
// ===== library types =====

TYPE "UDT_AO"
   STRUCT
      In : Real;   // Входное значение для вывода
      Par_max : Real := 100.0;   // Максимальное значение шкалы
      Par_min : Real;   // Минимальное занчение шкалы
      RezCh : Bool;   // В true если канал резервный
      Out : Int;   // Обработанное занчение на выход модуля
   END_STRUCT;
END_TYPE

TYPE "UDT_DI"
VERSION : 0.1
   STRUCT
      ReservChannel : Bool;   // Признак резервного бита
      Value : Bool;   // Выходное значение
      Invert : Bool;   // Инверсия
      In_Value : Bool;   // Входное значение
      Simulate : Bool;   // Симуляция
      Sim_Value : Bool;   // Значение симуляции
   END_STRUCT;
END_TYPE

TYPE "UDT_AI"
VERSION : 0.1
   STRUCT
      Raw_in : Int;   // Код АЦП - входное значение с модуля / Входной сигнал от модуля
      Out_value : Real;   // Масштабированное значение / Выходной преобразованный сигнал
      Field_value : Real;   // Значение тока (напряжения) с датчика
      Value_hi_scale : Int := 100;   // Максимальное физическое значение / Верняя шкала
      Value_lo_scale : Int;   // Минимальное физическое значение / Нижняя жкала
      Hihi_limit : Real;   // Значение верхней аварийной границы / ВАУ
      Hi_limit : Real;   // Значение верхней предупредительной границы / ВПУ
      Lo_limit : Real;   // Значение нижней предупредительной границы / НПУ
      Lolo_limit : Real;   // Значение нижней аварийной границы / НАУ
      Simulate_In : Real;   // Заданное значение симуляции / Значение симуляции
      Raw_lo_scale : Int := 5530;   // Код АЦП - нижняя граница значения
      Raw_hi_scale : Int := 27648;   // Код АЦП - верхняя граница значения
      Raw_lo_error : Int := 4838;   // Код АЦП - граница обрыва
      Raw_hi_error : Int := 28000;   // Код АЦП - граница короткого замыкания
      Field_lo_scale : Real := 4.0;   // Минимальное значение тока (напряжения)
      Field_hi_scale : Real := 20.0;   // Максимальное значение тока (напряжения)
      Digital_in : Real;   // Входное масштабированное значение
      RezervChannel : Bool;   // Признак резервного канала
      En_Digital_in : Bool;   // Разрешение - вход для значения Real вместо Int (Word)
      Simulate : Bool;   // Разрешение - режим симуляции / Признак цимуляции
      Hihi_enable : Bool;   // Разрешение - обработка сигнала Hihi / Активация ВАУ
      Hi_enable : Bool;   // Разрешение - обработка сигнала Hi / Активация ВПУ
      Lo_enable : Bool;   // Разрешение - обработка сигнала Lo / Активация НПУ
      Lolo_enable : Bool;   // Разрешение - обработка сигнала Lolo / Активация НАУ
      Hihi_act : Bool;   // Флаг - значение в верхней аварийной зоне / Сработка ВАУ
      Hi_act : Bool;   // Флаг - значение в верхней предупредительной зоне / Сработка ВПУ
      Lo_act : Bool;   // Флаг - значение в верхней предупредительной зоне / Сработка НПУ
      Lolo_act : Bool;   // Флаг - значение в нижней аварийной зоне / Сработка НАУ
      Lo_raw : Bool;   // Флаг - обрыв / Обрыв
      Hi_raw : Bool;   // Флаг - короткое замыкание / КЗ
      Alarm : Bool;   // Флаг - значение в аварийной зоне / Авария
      Warning : Bool;   // Флаг - значение в предупредительной зоне / Предупреждение
      Nominal : String := 'mm';   // Размерность един. изм.
   END_STRUCT;
END_TYPE

TYPE "UDT_IM"
   STRUCT
      SO : Bool;   // Состояние вкл/открыто
      SC : Bool;   // Состояние откл/закрыто
      SA : Bool;   // Состояние авария
      DU : Bool;   // Состояние дистанционное управление
      MU : Bool;   // Состояние местное управление
      Q_CO : Bool;   // Команда вкл/открыть
      Q_CS : Bool;   // Команда откл/закрыть
      B_CO : Bool;   // Команда открыть/вклюсить по алгоритму
      B_CS : Bool;   // Команда закрыть/выключить по алгоритму
      HMI_CO : Bool;   // Команда открыть/включить от ВУ
      HMI_CS : Bool;   // Команда закрыть/отключить от ВУ
      I_REP : Bool;   // Команда ремонт
      Q_REP : Bool;   // Выход команды ремонт
      Load : Int;   // Значение нагрузки
      TON_PT : Time := T#60000ms;
      TON_ET : Time;
      TON_IN : Bool;
      TON_Q : Bool;
   END_STRUCT;
END_TYPE

// folder: AI

FUNCTION "Proc_AI" : Void   // FC100, SCL
{ S7_Optimized_Access := 'TRUE' }
AUTHOR : SybCom
VERSION : 0.1
   VAR_TEMP
      i : Int;
      j : Int;
      Out_scaled : Real;
      AVG_Value : Real;
      Summ_Massive : Real;
      Result : Int;
      NumAnalog : Int;
      Dtl_now : DTL;
      One_sec_on : Bool;
      H_msec_on : Bool;
      AI_ACP_REAL : Real;
      MAX_ACP_REAL : Real;
      MIN_ACP_REAL : Real;
   END_VAR
BEGIN
   //AUTHOR: frozi2
   //DESC: Блок входного аналогового сигнала

   // Блок инициализации данных
   //2A1.3
   (*
   "Data_AI".Data[1].Raw_in := "AI1";//"PT-10"; //Давление сжатого воздуха
   "Data_AI".Data[2].Raw_in := "AI2";//"PT-01"; //Разрежение до РФ
   "Data_AI".Data[3].Raw_in := "AI3";//"PT-02"; //Разрежение после РФ
   "Data_AI".Data[4].Raw_in := "TT-01"; //Температура газа перед клапаном ав. подсоса
   "Data_AI".Data[5].Raw_in := "TT-02"; //Температура газа перед РФ
   "Data_AI".Data[6].Raw_in := "QT-101"; //Запыленность газа
   "Data_AI".Data[7].Raw_in := "FT-101"; //Расход газа
   "Data_AI".Data[8].Raw_in := "TT-03"; //Температура газа на выходе
   *)
   //2A1.4
   //"Data_AI".Data[9].Raw_in  := "2A1_4_AI_00"; //Давление воды 
   //"Data_AI".Data[10].Raw_in := "2A1_4_AI_01"; //Давление до 
   //"Data_AI".Data[11].Raw_in := "2A1_4_AI_02"; //Давление после 
   //"Data_AI".Data[12].Raw_in := "2A1_4_AI_03"; //Резерв
   //"Data_AI".Data[13].Raw_in := "2A1_4_AI_04"; //Резерв
   //"Data_AI".Data[14].Raw_in := "2A1_4_AI_05"; //Резерв
   //"Data_AI".Data[15].Raw_in := "2A1_4_AI_06"; //Резерв
   //"Data_AI".Data[16].Raw_in := "2A1_4_AI_07"; //Резерв
   (*
   FOR #i := 1 TO "Data_AI".Num_AI DO
       IF (#i > 4 AND #i < 9) OR #i > 11 THEN
           "Data_AI".Data[#i].RezervChannel := TRUE;
       ELSE
           "Data_AI".Data[#i].RezervChannel := FALSE;
       END_IF;
   END_FOR;
   *)

   //для расшифровки кода АЦП


   // Обработка сигналов
   FOR #i := 1 TO "Data_AI".Num_AI DO
     // Если канал не резервный
       IF NOT "Data_AI".Data[#i].RezervChannel THEN

           // Приведение к другому типу для удобства вычислений
           #AI_ACP_REAL := DINT_TO_REAL(WORD_TO_DINT("Data_AI".Data[#i].Raw_in));   // Перевод из WORD в REAL значение с АЦП входа
           #MAX_ACP_REAL := DINT_TO_REAL(WORD_TO_DINT("Data_AI".Data[#i].Value_hi_scale)); // Перевод из WORD в REAL Шкалы макс.
           #MIN_ACP_REAL := DINT_TO_REAL(WORD_TO_DINT("Data_AI".Data[#i].Value_lo_scale)); // Перевод из WORD в REAL Шкалы мин.

           //Масштабирование величин
           //Токовое значение с датчика   
           "Data_AI".Data[#i].Field_value := (("Data_AI".Data[#i].Field_hi_scale - "Data_AI".Data[#i].Field_lo_scale) / ("Data_AI".Data[#i].Raw_hi_scale - "Data_AI".Data[#i].Raw_lo_scale)) *
           ("Data_AI".Data[#i].Raw_in - "Data_AI".Data[#i].Raw_lo_scale) + "Data_AI".Data[#i].Field_lo_scale;

           //Физическое значение с датчика
           #Out_scaled := (#MAX_ACP_REAL - #MIN_ACP_REAL) / ("Data_AI".Data[#i].Raw_hi_scale - "Data_AI".Data[#i].Raw_lo_scale) *
           (#AI_ACP_REAL - "Data_AI".Data[#i].Raw_lo_scale) + #MIN_ACP_REAL;



       // Полученный сигнал уже масштабирован
       IF "Data_AI".Data[#i].En_Digital_in THEN
         #Out_scaled := "Data_AI".Data[#i].Digital_in;
       END_IF;
       // Симуляция выходной величины
       IF "Data_AI".Data[#i].Simulate THEN
         #Out_scaled := "Data_AI".Data[#i].Simulate_In;
       END_IF;
       // Усреднение и нижняя отсечка (удалено из DB)    
       (*  

       //Запоминание времени
       #Result := RD_LOC_T(#Dtl_now);
       //Счетчик для усреднения величины
       if TOD_TO_DINT(DTL_TO_TOD(#Dtl_now)) - TOD_TO_DINT(DTL_TO_TOD("DataHelpAI".Data[i].Dtl_h_msec)) >
          INT_TO_DINT("DataHelpAI".Data[i].Bal_time) * 100 then
         #H_msec_on := True;
       end_if;
       //Усреднение величины ведется с кратностью в 100 мс.
       if #H_msec_on then
         #Result := RD_LOC_T("DataHelpAI".Data[i].Dtl_h_msec);
         #H_msec_on := False;
         //Запись в массив ведется циклично
         "DataHelpAI".Data[i].Massive_point := "DataHelpAI".Data[i].Massive_point + 1;  
         if "DataHelpAI".Data[i].Massive_point > 9 then
           "DataHelpAI".Data[i].Massive_point := 0;
         end_if;
         //Сохранение величины в массиве
         "DataHelpAI".Data[i].Output_Massive["DataHelpAI".Data[i].Massive_point] := #Out_scaled;  
       end_if;
       #AVG_Value := 0;
       if "DataHelpAI".Data[i].Bal_time > 0 then
         #Summ_Massive := 0;
         for #j := 0 to 9 do
           #Summ_Massive := #Summ_Massive + "DataHelpAI".Data[i].Output_Massive[#j];
         end_for;
         #AVG_Value := #Summ_Massive / 10;
         #Out_scaled := #AVG_Value;
       end_if;
       //Проверка на зону нечувствительности 
       if ABS("DataHelpAI".Data[i].Previos_val - #Out_scaled) < "DataHelpAI".Data[i].Value_db then
         #Out_scaled := "DataHelpAI".Data[i].Previos_val;
       end_if;
       //Проверка на нижнюю отсечку  
       if (#Out_scaled < "DataHelpAI".Data[i].Lo_cutoff) & "DataHelpAI".Data[i].Lo_cut_enable then
         #Out_scaled := "DataHelpAI".Data[i].Lo_cutoff;
       end_if;
   *)



       // Формирование аварий  
       // Обрыв  
       IF ("Data_AI".Data[#i].Raw_in <= "Data_AI".Data[#i].Raw_lo_error) AND
         NOT "Data_AI".Data[#i].Simulate THEN
         "Data_AI".Data[#i].Lo_raw := True;
         #Out_scaled := "Data_AI".Data[#i].Value_lo_scale;
       ELSE
         "Data_AI".Data[#i].Lo_raw := False;
       END_IF;

       // КЗ датчика
       IF ("Data_AI".Data[#i].Raw_in >= "Data_AI".Data[#i].Raw_hi_error) AND
         NOT "Data_AI".Data[#i].Simulate THEN
         "Data_AI".Data[#i].Hi_raw := True;
         #Out_scaled := "Data_AI".Data[#i].Value_hi_scale;
       ELSE
         "Data_AI".Data[#i].Hi_raw := False;
       END_IF;

       // Нижняя аварийная зона
       IF #Out_scaled < "Data_AI".Data[#i].Lolo_limit AND
           "Data_AI".Data[#i].Lolo_enable AND NOT "Data_AI".Data[#i].Lo_raw THEN
           "Data_AI".Data[#i].Lolo_act := True;
       ELSE
           "Data_AI".Data[#i].Lolo_act := False;
       END_IF;

       // Нижняя предупредительная зона
       IF #Out_scaled < "Data_AI".Data[#i].Lo_limit AND NOT "Data_AI".Data[#i].Lolo_act AND
           "Data_AI".Data[#i].Lo_enable AND NOT "Data_AI".Data[#i].Lo_raw THEN
           "Data_AI".Data[#i].Lo_act := True;
       ELSE
           "Data_AI".Data[#i].Lo_act := False;
       END_IF;
       // Верхняя предупредительная зона
       IF #Out_scaled > "Data_AI".Data[#i].Hi_limit AND NOT "Data_AI".Data[#i].Hihi_act AND
           "Data_AI".Data[#i].Hi_enable AND NOT "Data_AI".Data[#i].Hi_raw THEN
           "Data_AI".Data[#i].Hi_act := True;
       ELSE
           "Data_AI".Data[#i].Hi_act := False;
       END_IF;

       // Верхняя аварийная зона
       IF #Out_scaled > "Data_AI".Data[#i].Hihi_limit AND
           "Data_AI".Data[#i].Hihi_enable AND NOT "Data_AI".Data[#i].Hi_raw THEN
           "Data_AI".Data[#i].Hihi_act := True;
       ELSE
           "Data_AI".Data[#i].Hihi_act := False;
       END_IF;

       // Определение флага предупреждения
       IF ("Data_AI".Data[#i].Hi_act OR "Data_AI".Data[#i].Lo_act) THEN
         "Data_AI".Data[#i].Warning := true;
       ELSE
         "Data_AI".Data[#i].Warning := false;
       END_IF;

       // Определение флага аварии
       IF "Data_AI".Data[#i].Hihi_act OR "Data_AI".Data[#i].Lolo_act  THEN
         "Data_AI".Data[#i].Alarm := true;
       ELSE
         "Data_AI".Data[#i].Alarm := false;
       END_IF;

       // Сохранение значения
       "Data_AI".Data[#i].Out_value := #Out_scaled;
     END_IF;
   END_FOR;
END_FUNCTION

// folder: AO

FUNCTION "Proc_AO" : Void   // FC102, SCL
{ S7_Optimized_Access := 'TRUE' }
VERSION : 0.1
   VAR_TEMP
      i : Int;
      Temp_out : Real;
   END_VAR
BEGIN
   //AUTHOR: frozi2
   //DESC: Блок выходного аналогового сигнала

   // Блок инициализации данных
   //2A1.3
   "Data_AO".Data[1].In := "AI1";//"PT-10"; //Давление сжатого воздуха
   "Data_AO".Data[2].In := "AI2";//"PT-01"; //Разрежение до РФ
   "Data_AO".Data[3].In := "AI3";//"PT-02"; //Разрежение после РФ
   "Data_AO".Data[4].In := "TT-01"; //Температура газа перед клапаном ав. подсоса
   "Data_AO".Data[5].In := "TT-02"; //Температура газа перед РФ
   "Data_AO".Data[6].In := "QT-101"; //Запыленность газа
   "Data_AO".Data[7].In := "FT-101"; //Расход газа
   "Data_AO".Data[8].In := "TT-03"; //Температура газа на выходе


   //Задействовать это часть для анализа резервных каналов и исключения их их опроса или принудительно
   //устанавливать переменную RezervChannel = 1, в Data_AO для каждого резервного канала
   (*
   FOR #i := 1 TO "Data_AI".Num_AO DO
       IF (#i > 4 AND #i < 9) OR #i > 11 THEN  //тут отредактировать по своим условиям
           "Data_AO".Data[#i].RezCh := TRUE;
       ELSE
           "Data_A0".Data[#i].RezCh := FALSE;
       END_IF;
   END_FOR;
   *)

   // Обработка сигналов
   FOR #i := 1 TO "Data_AO".Num_AO DO

       #Temp_out := ((27648.0 - 0.0)*("Data_AO".Data[#i].In - "Data_AO".Data[#i].Par_min))/("Data_AO".Data[#i].Par_max - "Data_AO".Data[#i].Par_min);

       // Если канал не резервный
       IF NOT "Data_AO".Data[#i].RezCh THEN

           // Сохранение значения
           "Data_AO".Data[#i].Out := DINT_TO_INT(REAL_TO_DINT(#Temp_out));

       END_IF;

   END_FOR;
END_FUNCTION

// folder: DI

FUNCTION "Proc_DI" : Void   // FC101, SCL
{ S7_Optimized_Access := 'TRUE' }
AUTHOR : SybCom
VERSION : 0.1
   VAR_TEMP
      i : Int;
      j : Int;
      TempValue : Bool;
      H_msec_on : Bool;
      Result : Int;
      Dtl_now : DTL;
      Summ_Massive : Real;
   END_VAR
BEGIN
   //AUTHOR: frozi2
   //DESC: Блок дискретного сигнала

   // Блок инициализации данных
   // 2A1
   "Data_DI".Data[1].In_Value := "LSA-11";  //Минимальный уровень бункера 1
   "Data_DI".Data[2].In_Value := "LSA-12";  //Верхний уровень бункера 1
   "Data_DI".Data[3].In_Value := "LSA-13";  //Минимальный уровень бункера 2
   "Data_DI".Data[4].In_Value := "LSA-14";  //Верхний уровень бункера 2
   "Data_DI".Data[5].In_Value := "LSA-15";  //Минимальный уровень бункера 3
   "Data_DI".Data[6].In_Value := "LSA-16";  //Верхний уровень бункера 3
   "Data_DI".Data[7].In_Value := "LSA-17";  //Минимальный уровень бункера 4
   "Data_DI".Data[8].In_Value := "LSA-18";  //Верхний уровень бункера 4
   "Data_DI".Data[9].In_Value := 0;  //Резерв
   "Data_DI".Data[10].In_Value := 0; //Резерв
   "Data_DI".Data[11].In_Value := 0; //Резерв
   "Data_DI".Data[12].In_Value := 0; //Резерв
   "Data_DI".Data[13].In_Value := 0; //Резерв
   "Data_DI".Data[14].In_Value := 0; //Резерв
   (*
   //2A1.5
   "Data_DI".Data[15].In_Value := "2A1_5_DI_00"; //Зд1 поз.7.2 - Открыта
   "Data_DI".Data[16].In_Value := "2A1_5_DI_01"; //Зд1 поз.7.2 - Закрыта
   "Data_DI".Data[17].In_Value := "2A1_5_DI_02"; //Зд1 поз.7.2 - Неисправность
   "Data_DI".Data[18].In_Value := "2A1_5_DI_03"; //Зд2 поз.7.2 - Открыта
   "Data_DI".Data[19].In_Value := "2A1_5_DI_04"; //Зд2 поз.7.2 - Закрыта
   "Data_DI".Data[20].In_Value := "2A1_5_DI_05"; //Зд2 поз.7.2 - Неисправность
   "Data_DI".Data[21].In_Value := "2A1_5_DI_06"; //Зд3 поз.7.2 - Открыта
   "Data_DI".Data[22].In_Value := "2A1_5_DI_07"; //Зд3 поз.7.2 - Закрыта
   "Data_DI".Data[23].In_Value := "2A1_5_DI_08"; //Зд3 поз.7.2 - Неисправность
   "Data_DI".Data[24].In_Value := "2A1_5_DI_09"; //УПОУ поз.7.2 - Исправен 1к
   "Data_DI".Data[25].In_Value := "2A1_5_DI_10"; //УПОУ поз.7.2 - ВТО 1к
   "Data_DI".Data[26].In_Value := "2A1_5_DI_11"; //Резерв
   "Data_DI".Data[27].In_Value := "2A1_5_DI_12"; //С2000-СП1 №1 - «Пожар в блоке» - поз.2.3
   "Data_DI".Data[28].In_Value := "2A1_5_DI_13"; //С2000-СП1 №1 - «Пожар в блоке» - поз.3.2
   "Data_DI".Data[29].In_Value := "2A1_5_DI_14"; //С2000-СП1 №1 - «Пожар в блоке» - поз.6.3(1)
   "Data_DI".Data[30].In_Value := "2A1_5_DI_15"; //С2000-СП1 №1 - «Пожар в блоке» - поз.6.3(2)

   //2A1.6
   "Data_DI".Data[31].In_Value := "2A1_6_DI_00"; //С2000-СП1 №2 - «Пожар»
   "Data_DI".Data[32].In_Value := "2A1_6_DI_01"; //С2000-СП1 №2 - «Неисправность»
   "Data_DI".Data[33].In_Value := "2A1_6_DI_02"; //Резерв
   "Data_DI".Data[34].In_Value := "2A1_6_DI_03"; //Резерв
   "Data_DI".Data[35].In_Value := "2A1_6_DI_04"; //Сигнал 20П - Несанкционированный вход
   "Data_DI".Data[36].In_Value := "2A1_6_DI_05"; //Сигнал 20П - Неисправность
   "Data_DI".Data[37].In_Value := "2A1_6_DI_06"; //Шкаф ШОС - Обобщенный сигнал несанкционированного входа
   "Data_DI".Data[38].In_Value := "2A1_6_DI_07"; //Шкаф ШОС - Неисправность
   "Data_DI".Data[39].In_Value := "2A1_6_DI_08"; //Состояние ЭЦН скважины 1.25
   "Data_DI".Data[40].In_Value := "2A1_6_DI_09"; //Состояние ЭЦН скважины 1.26
   "Data_DI".Data[41].In_Value := "2A1_6_DI_10"; //Состояние ЭЦН скважины 1.27
   "Data_DI".Data[42].In_Value := "2A1_6_DI_11"; //Состояние ЭЦН скважины 1.28
   "Data_DI".Data[43].In_Value := "2A1_6_DI_12"; //Состояние ЭЦН скважины 1.29
   "Data_DI".Data[44].In_Value := "2A1_6_DI_13"; //Состояние ЭЦН скважины 1.30
   "Data_DI".Data[45].In_Value := "2A1_6_DI_14"; //Состояние ЭЦН скважины 1.31
   "Data_DI".Data[46].In_Value := "2A1_6_DI_15"; //Состояние ЭЦН скважины 1.32

   //2A1.7
   "Data_DI".Data[47].In_Value := "2A1_7_DI_00"; //Состояние ЭЦН скважины 1.33
   "Data_DI".Data[48].In_Value := "2A1_7_DI_01"; //Состояние ЭЦН скважины 1.34
   "Data_DI".Data[49].In_Value := "2A1_7_DI_02"; //Состояние ЭЦН скважины 1.35
   "Data_DI".Data[50].In_Value := "2A1_7_DI_03"; //Состояние ЭЦН скважины 1.36
   "Data_DI".Data[51].In_Value := "2A1_7_DI_04"; //Состояние ЭЦН скважины 1.37
   "Data_DI".Data[52].In_Value := "2A1_7_DI_05"; //Состояние ЭЦН скважины 1.38
   "Data_DI".Data[53].In_Value := "2A1_7_DI_06"; //Состояние ЭЦН скважины 1.39
   "Data_DI".Data[54].In_Value := "2A1_7_DI_07"; //Состояние ЭЦН скважины 1.40
   "Data_DI".Data[55].In_Value := "2A1_7_DI_08"; //Состояние ЭЦН скважины 1.41
   "Data_DI".Data[56].In_Value := "2A1_7_DI_09"; //Состояние ЭЦН скважины 1.42
   "Data_DI".Data[57].In_Value := "2A1_7_DI_10"; //Состояние ЭЦН скважины 1.43
   "Data_DI".Data[58].In_Value := "2A1_7_DI_11"; //Резерв
   "Data_DI".Data[59].In_Value := "2A1_7_DI_12"; //Резерв
   "Data_DI".Data[60].In_Value := "2A1_7_DI_13"; //Резерв
   "Data_DI".Data[61].In_Value := "2A1_7_DI_14"; //Резерв
   "Data_DI".Data[62].In_Value := "2A1_7_DI_15"; //Резерв

   // Заклинивание в Орион+
   "Data_DI".Data[63].In_Value := WORD_TO_INT("Data_Valve".Data[1].Alarm) > 1; // Зд1 УПОУ поз.7.2
   "Data_DI".Data[64].In_Value := WORD_TO_INT("Data_Valve".Data[2].Alarm) > 1; // Зд2 УПОУ поз.7.2
   "Data_DI".Data[65].In_Value := WORD_TO_INT("Data_Valve".Data[3].Alarm) > 1; // Зд3 УПОУ поз.7.2

   // Автоматический режим в Орион+
   "Data_DI".Data[66].In_Value := "Data_Valve".Data[1].Mode_auto; //Зд1 УПОУ поз.7.2
   "Data_DI".Data[67].In_Value := "Data_Valve".Data[2].Mode_auto; //Зд2 УПОУ поз.7.2
   "Data_DI".Data[68].In_Value := "Data_Valve".Data[3].Mode_auto; //Зд3 УПОУ поз.7.2

   // Сигналы ПАЗ для Орион
   "Data_DI".Data[69].In_Value := "Data_AI".Data[10].Hihi_act;
   "Data_DI".Data[70].In_Value := "Data_AI".Data[10].Lolo_act;
   "Data_DI".Data[71].In_Value := "Data_AI".Data[11].Hihi_act;
   "Data_DI".Data[72].In_Value := "Data_AI".Data[11].Lolo_act;

   // Сигналы ПАЗ для Орион(Состояние вкл\выкл)
   "Data_DI".Data[73].In_Value := "Data_AI".Data[10].Hihi_enable;
   "Data_DI".Data[74].In_Value := "Data_AI".Data[10].Lolo_enable;
   "Data_DI".Data[75].In_Value := "Data_AI".Data[11].Hihi_enable;
   "Data_DI".Data[76].In_Value := "Data_AI".Data[11].Lolo_enable;
   *)
   (*
   //Отключение в обработке неиспользуемых дискретных входов
   FOR #i := 1 TO "Data_DI".Num_DI DO
       IF (#i > 6 AND #i < 9) OR (#i > 10 AND #i < 15) OR #i = 26 OR (#i > 32 AND #i < 35) OR (#i > 57 AND #i < 63) OR #i > 76 THEN
           "Data_DI".Data[#i].ReservChannel := TRUE;
       ELSE
           "Data_DI".Data[#i].ReservChannel := FALSE;
       END_IF;
   END_FOR;
   *)

   FOR #i := 1 TO "Data_DI".Num_DI DO
     IF NOT "Data_DI".Data[#i].ReservChannel THEN
       #TempValue := False;
       // Эмитация значения 
       IF "Data_DI".Data[#i].Simulate THEN
         #TempValue := "Data_DI".Data[#i].Sim_Value;
       ELSE
         #TempValue := "Data_DI".Data[#i].In_Value;
       END_IF;

       // Инвертирование значения
       #TempValue := #TempValue XOR "Data_DI".Data[#i].Invert;

       // Убрал фильтрацию 
       (*
       #Result := RD_LOC_T(#Dtl_now);                                                          // Запоминание времени

       if TOD_TO_DINT(DTL_TO_TOD(#Dtl_now)) - TOD_TO_DINT(DTL_TO_TOD("Data_DI".Data[#i].Dtl_h_msec)) >
           INT_TO_DINT("Data_DI".Data[#i].Filter_Time_hms) * 25 then                         // Счетчик для определения скачка величины
           #H_msec_on := true;
       end_if;

       if #H_msec_on then
           #Result := RD_LOC_T("Data_DI".Data[#i].Dtl_h_msec);
           "Data_DI".Data[#i].Massive_point := "Data_DI".Data[#i].Massive_point + 1;  //Запись в массив ведется циклично
           if "Data_DI".Data[#i].Massive_point > 9 then
               "Data_DI".Data[#i].Massive_point := 0;
           end_if;
           "Data_DI".Data[#i].Output_Massive["Data_DI".Data[#i].Massive_point] := #TempValue;  //Сохранение величины в массиве
           #H_msec_on := false;
       end_if;

       if "Data_DI".Data[#i].Filter_On then  //Фильтр позволит отбросить случайные срабатывания на канале DI
           #Summ_Massive := 0;
           for #j := 0 to 9 do
               if "Data_DI".Data[#j].Output_Massive[#j] = true then
                   #Summ_Massive := #Summ_Massive + 1;
               end_if;
           end_for;
           if #Summ_Massive > 5 then  //Выходное значение будет истинным, только при наборе более половины массива значений
               #TempValue := true;
           else
               #TempValue := false;
           end_if;
       end_if;
       *)
       "Data_DI".Data[#i].Value := #TempValue;
     END_IF;
   END_FOR;
END_FUNCTION

// folder: DO

FUNCTION "Proc_DO" : Void   // FC103, SCL
{ S7_Optimized_Access := 'TRUE' }
VERSION : 0.1
BEGIN
   //Author: frozi2
   //Deck: Блок дискретных выходов

   // // Отключение вводов по пожару
   // IF NOT "Block_Temp".Temp_2_3_3_2 AND "Block_Temp".On_2_3_3_2 THEN //Если нет аварии, тогда до отработает по сигналу пожаров
   //     "Data_DO".Data[13] := "Data_DI".Data[27].Value OR "Data_DI".Data[28].Value; // Отключение поз.2.3,3.2 при пожаре в поз.2.3,поз.3.2 //собрана схема таким образом, что АГЗУ питается от ЩСН
   //     "Data_DO".Data[14] := "Data_DI".Data[27].Value OR "Data_DI".Data[28].Value; // Отключение поз.2.3,3.2 при пожаре в поз.2.3,поз.3.2 //собрана схема таким образом, что АГЗУ питается от ЩСН
   //     "Data_DO".Data[11] := "Data_DI".Data[28].Value;  // Отключение поз.2.3,3.2 при пожаре в поз.2.3,поз.3.2 //собрана схема таким образом, что АГЗУ питается от ЩСН
   //     "Data_DO".Data[12] := "Data_DI".Data[28].Value;  // Отключение поз.2.3,3.2 при пожаре в поз.2.3,поз.3.2 //собрана схема таким образом, что АГЗУ питается от ЩСН
   //     "Block_Temp".Temp_2_3_3_2 := ("Data_DO".Data[13] AND "Data_DO".Data[14]) OR ("Data_DO".Data[11] AND "Data_DO".Data[12]);
   // END_IF;

   // IF "Block_Temp".Temp_2_3_3_2 THEN//Если авария возникла, тогда так как до отработали ранее сбрасываем до, чтобы не сгорели расцепители
   //     "Data_DO".Data[13] := False; // Отключение поз.2.3,3.2 при пожаре в поз.2.3,поз.3.2 //собрана схема таким образом, что АГЗУ питается от ЩСН
   //     "Data_DO".Data[14] := False; // Отключение поз.2.3,3.2 при пожаре в поз.2.3,поз.3.2 //собрана схема таким образом, что АГЗУ питается от ЩСН
   //     "Data_DO".Data[11] := False; // Отключение поз.2.3,3.2 при пожаре в поз.2.3,поз.3.2 //собрана схема таким образом, что АГЗУ питается от ЩСН
   //     "Data_DO".Data[12] := False; // Отключение поз.2.3,3.2 при пожаре в поз.2.3,поз.3.2 //собрана схема таким образом, что АГЗУ питается от ЩСН
   //     "Block_Temp".Temp_2_3_3_2 := "Data_DI".Data[27].Value OR "Data_DI".Data[28].Value;
   // END_IF;
   // 
   //2А1
   //"Out0" := "Data_DO".Data[1];  //Контроль 1к
   //"Out1" := "Data_DO".Data[2];  //УП2 - Сброс 1к
   //"Out2" := "Data_DO".Data[3];  //ДЕ поз.5.4
   //"Out3" := "Data_DO".Data[4];  //ДЕ поз.5.4
   //"Out4" := "Data_DO".Data[5];  //ДЕ поз.5.3
   //"Out5" := "Data_DO".Data[6];  //ДЕ поз.5.3
   //"Out6" := "Data_DO".Data[7];  //Резерв
   //"Out7" := "Data_DO".Data[8];  //Резерв
END_FUNCTION

// folder: IM

FUNCTION "Proc_IM" : Void   // FC105, SCL
{ S7_Optimized_Access := 'TRUE' }
VERSION : 0.1
   VAR_TEMP
      i : Int;
   END_VAR
   VAR CONSTANT
      Time_run : Time := T#60000ms;
   END_VAR
BEGIN
   //AUTHOR: frozi2
   //DESC: Блок обработки исполниельных механизмов

   // Блок инициализации данных и просто памятка по сигналам
   // 
   //"Data_IM".Data[#i].SO := "VIB_1M1_SO"; //состояние открыт/включен
   //"Data_IM".Data[#i].SC := NOT "VIB_1M1_SO"; //состояние закрыт/отключен
   //"Data_IM".Data[#i].SA := "VIB_1M1_SA"; //состояние авария
   //"Data_IM".Data[#i].DU := "VIB_1M1_DU"; //режим дистанц. управление
   //"Data_IM".Data[#i].MU := NOT "VIB_1M1_DU"; //режим мест. управление
   //"Data_IM".Data[#i].Q_CO := "VIB_1M1_COCS"; //команда открыть/вкл
   //"Data_IM".Data[#i].Q_CS := NOT "VIB_1M1_COCS"; //команда закрыть/откл
   //"Data_IM".Data[#i].B_CO:= 0; //Команда открыть/вклюсить по алгоритму
   //"Data_IM".Data[#i].B_CS:= 0; //Команда закрыть/выключить по алгоритму
   //"Data_IM".Data[#i].HMI_CO:= 0; //команда управления с HMI открыть/вкл
   //"Data_IM".Data[#i].HMI_CS:= 0; //команда управления с HMI  закрыть/откл
   //"Data_IM".Data[#i].I_REP:= 0; //Команда ремонт
   //"Data_IM".Data[#i].Q_REP:= 0; //Выход команды ремонт
   //"Data_IM".Data[#i].Load := 0; //нагрузка двигателя (опционально)

   //Перебор всех исполнительных механихмов (ИМ)
   FOR #i:= 1 TO "Data_IM".Num_IM DO

       //Инициализация времени для таймера, устанавливаем на 60 сек
       "Data_IM".Data[#i].TON_ET:= #Time_run;

       //Формирование состояние авария
       IF    ("Data_IM".Data[#i].SO      //состояние открыт/включен
           AND "Data_IM".Data[#i].TON_Q )
           OR  "Data_IM".Data[#i].TON_Q//таймер досчитал
       THEN
           "Data_IM".Data[#i].SA := 1;
       ELSE
           "Data_IM".Data[#i].SA := 0;
       END_IF;


       //Формирование команды открыть/включить
       IF (("Data_IM".Data[#i].B_CO        //Команда открыть/вклюсить по алгоритму
         OR "Data_IM".Data[#i].HMI_CO)     //команда управления с HMI открыть/вкл

           AND NOT "Data_IM".Data[#i].SA         //не аварии
           AND NOT "Data_IM".Data[#i].SO         //нет состояни открыт/включен
           AND NOT "Data_IM".Data[#i].Q_REP      //нет ремонта
           AND     "Data_IM".Data[#i].DU)        //режим дистанционный
       THEN
           "Data_IM".Data[#i].Q_CO := 1;
           "Data_IM".Data[#i].Q_CS := 0;
           "Data_IM".Data[#i].TON_IN := 1; //запускаем таймер на 60 сек
       END_IF;

       //Формирование команды закрыть/отключить
       IF (("Data_IM".Data[#i].B_CS      //Команда открыть/вклюсить по алгоритму
           OR "Data_IM".Data[#i].HMI_CS)     //команда управления с HMI открыть/вкл

           AND NOT "Data_IM".Data[#i].SA         //не аварии
           AND     "Data_IM".Data[#i].SO         //нет состояни открыт/включен
           AND NOT "Data_IM".Data[#i].Q_REP      //нет ремонта
           AND     "Data_IM".Data[#i].DU)        //режим дистанционный
       THEN
           "Data_IM".Data[#i].Q_CS := 1;
           "Data_IM".Data[#i].Q_CO := 0;
           "Data_IM".Data[#i].TON_IN := 1; //запускаем таймер на 60 сек
       END_IF;


       //Часть сброса таймера
       IF      ("Data_IM".Data[#i].SO AND ("Data_IM".Data[#i].B_CO OR "Data_IM".Data[#i].HMI_CO))    //Если открыт/включен и есть команда на открыть по алгоритму и от HMI
           OR  (NOT "Data_IM".Data[#i].SO AND ("Data_IM".Data[#i].B_CS OR "Data_IM".Data[#i].HMI_CS))//Если не открыт и есть команда на закрыть по алгоритму и от HMI
           OR  "Data_IM".Data[#i].SA //Если есть авария
       THEN
           "Data_IM".Data[#i].TON_IN:= 0; //сбрасываем таймер;
       END_IF;

       //Просто вызов блока таймера с задержкой на отключение для расчета времени открытия/закрытия, включения/отключения
       "Data_IM".Timer_run[#i].TON(IN :="Data_IM".Data[#i].TON_IN,
                                   PT := "Data_IM".Data[#i].TON_PT,
                                   Q => "Data_IM".Data[#i].TON_Q,
                                   ET => "Data_IM".Data[#i].TON_ET);

   END_FOR;
END_FUNCTION

// ===== library: MasterCopy "Data_IM" =====

// folder: IM

DATA_BLOCK "Data_IM"   // DB105
{ S7_Optimized_Access := 'TRUE' }
VERSION : 0.1
   VAR
      Data : Array[1..128] of "UDT_IM";
      Timer_run : Array[1..128] of IEC_TIMER;
      Num_IM : Int := 128;
   END_VAR
BEGIN
END_DATA_BLOCK

// ===== library: MasterCopy "Data_DO" =====

// folder: DO

DATA_BLOCK "Data_DO"   // DB103
{ S7_Optimized_Access := 'FALSE' }
AUTHOR : SybCom
VERSION : 3.0
   VAR
      Data : Array[1..128] of Bool;
      Num_DO : Int := 128;
   END_VAR
BEGIN
END_DATA_BLOCK

// ===== library: MasterCopy "Data_DI" =====

// folder: DI

DATA_BLOCK "Data_DI"   // DB101
{ S7_Optimized_Access := 'FALSE' }
VERSION : 0.1
   VAR
      Data : Array[1..128] of "UDT_DI";
      Num_DI : Int := 128;
   END_VAR
BEGIN
END_DATA_BLOCK

// ===== library: MasterCopy "Data_AI" =====

// folder: AI

DATA_BLOCK "Data_AI"   // DB100
{ S7_Optimized_Access := 'FALSE' }
AUTHOR : frozi2
VERSION : 3.0
   VAR
      Data : Array[1..64] of "UDT_AI";
      Num_AI : Int := 64;
   END_VAR
BEGIN
   Data[1].Value_hi_scale := 100;
   Data[1].Hihi_limit := 95.0;
   Data[1].Hi_limit := 90.0;
   Data[1].Hihi_enable := 1;
   Data[1].Hi_enable := 1;
   Data[2].Value_hi_scale := 100;
   Data[2].Hihi_limit := 1.65;
   Data[2].Hi_limit := 1.5;
   Data[2].Hihi_enable := false;
   Data[2].Hi_enable := false;
   Data[3].Value_hi_scale := 100;
   Data[3].Hihi_limit := 0.0;
   Data[3].Hi_limit := 10.0;
   Data[3].Hihi_enable := false;
   Data[3].Hi_enable := false;
   Data[4].Value_hi_scale := 100;
   Data[4].Hihi_limit := 1.65;
   Data[4].Hi_limit := 1.5;
   Data[4].Hihi_enable := false;
   Data[4].Hi_enable := false;
   Data[1].Lolo_limit := 5.0;
   Data[2].Lolo_limit := 0.0;
   Data[3].Lolo_limit := 5.0;
   Data[4].Lolo_limit := 0.0;
   Data[1].Lo_limit := 10.0;
   Data[2].Lo_limit := 0.5;
   Data[4].Lo_limit := 0.5;
   Data[3].Lo_limit := 6.0;
   Data[9].Value_hi_scale := 100;
   Data[9].Lolo_limit := 137.66;
   Data[10].Raw_in := 0;
   Data[10].Out_value := 0.0;
   Data[10].Field_value := 0.0;
   Data[10].Value_hi_scale := 100;
   Data[10].Value_lo_scale := 0;
   Data[10].Hihi_limit := 40.79;
   Data[10].Hi_limit := 39.77;
   Data[10].Lo_limit := 0.0;
   Data[10].Lolo_limit := 10.2;
   Data[10].Simulate_In := 0.0;
   Data[10].Raw_lo_scale := 5530;
   Data[10].Raw_hi_scale := 27648;
   Data[10].Raw_lo_error := 4838;
   Data[10].Raw_hi_error := 28000;
   Data[10].Field_lo_scale := 4.0;
   Data[10].Field_hi_scale := 20.0;
   Data[10].Digital_in := 0.0;
   Data[10].RezervChannel := false;
   Data[10].En_Digital_in := false;
   Data[10].Simulate := false;
   Data[10].Hihi_enable := false;
   Data[10].Hi_enable := false;
   Data[10].Lo_enable := false;
   Data[10].Lolo_enable := false;
   Data[10].Hihi_act := false;
   Data[10].Hi_act := false;
   Data[10].Lo_act := false;
   Data[10].Lolo_act := false;
   Data[10].Lo_raw := false;
   Data[10].Hi_raw := false;
   Data[10].Alarm := false;
   Data[10].Warning := false;
   Data[11].Raw_in := 0;
   Data[11].Out_value := 0.0;
   Data[11].Field_value := 0.0;
   Data[11].Value_hi_scale := 50;
   Data[11].Value_lo_scale := 0;
   Data[11].Hihi_limit := 40.79;
   Data[11].Hi_limit := 39.77;
   Data[11].Lo_limit := 0.0;
   Data[11].Lolo_limit := 10.2;
   Data[11].Simulate_In := 0.0;
   Data[11].Raw_lo_scale := 5530;
   Data[11].Raw_hi_scale := 27648;
   Data[11].Raw_lo_error := 4838;
   Data[11].Raw_hi_error := 28000;
   Data[11].Field_lo_scale := 4.0;
   Data[11].Field_hi_scale := 20.0;
   Data[11].Digital_in := 0.0;
   Data[11].RezervChannel := false;
   Data[11].En_Digital_in := false;
   Data[11].Simulate := false;
   Data[11].Hihi_enable := false;
   Data[11].Hi_enable := false;
   Data[11].Lo_enable := false;
   Data[11].Lolo_enable := false;
   Data[11].Hihi_act := false;
   Data[11].Hi_act := false;
   Data[11].Lo_act := false;
   Data[11].Lolo_act := false;
   Data[11].Lo_raw := false;
   Data[11].Hi_raw := false;
   Data[11].Alarm := false;
   Data[11].Warning := false;
   Data[1].Lo_enable := 1;
   Data[1].Lolo_enable := 1;
   Data[1].Value_lo_scale := 0;
END_DATA_BLOCK

// ===== library: MasterCopy "Data_AO" =====

// folder: AO

DATA_BLOCK "Data_AO"   // DB102
{ S7_Optimized_Access := 'TRUE' }
VERSION : 0.1
   VAR
      Data : Array[1..16] of "UDT_AO";
      Num_AO : Int := 16;
   END_VAR
BEGIN
   Data[1].Par_min := 0.0;
   Data[2].Par_min := 0.0;
END_DATA_BLOCK

(* ===== HMI "HMI_RT_1" =====

ScreenModuleEditorView "FP_AI" 330x478
   IOField "I/O field_1" at 90,12 size 166x49; FormatPattern 999999
      ProcessValue <- "Data_AI.Out_value"
   TextField "Text field_1" at 263,22 size 45x29; Text 'мм'
   TextField "VAU" at 5,12 size 80x49; Text 'ВАУ'
      Visibility <- "Data_AI.Hihi_act"
   TextField "HAU" at 5,12 size 80x49; Text 'НАУ'
      Visibility <- "Data_AI.Lolo_act"
   TextField "VPU" at 5,12 size 80x49; Text 'ВПУ'
      Visibility <- "Data_AI.Hi_act"
   TextField "NPU" at 5,12 size 80x49; Text 'НПУ'
      Visibility <- "Data_AI.Lo_act"
   Switch "VAU_enable" at 35,72 size 135x50; TextOn 'Вкл'; CaptionText 'Активация ВАУ'; TextOff 'Откл'
      ProcessValue <- "Data_AI.Hihi_enable"
   Switch "VPU_enable" at 35,135 size 135x50; TextOn 'Вкл'; CaptionText 'Активация ВПУ'; TextOff 'Откл'
      ProcessValue <- "Data_AI.Hi_enable"
   Switch "NPU_enable" at 34,198 size 136x50; TextOn 'Вкл'; CaptionText 'Активация НПУ'; TextOff 'Откл'
      ProcessValue <- "Data_AI.Lo_enable"
   Switch "NAU_enable" at 35,262 size 135x50; TextOn 'Вкл'; CaptionText 'Активация НАУ'; TextOff 'Откл'
      ProcessValue <- "Data_AI.Lolo_enable"
   IOField "I/O field_2" at 189,86 size 121x37; FormatPattern 999999
      ProcessValue <- "Data_AI.Hihi_limit"
   IOField "I/O field_3" at 189,148 size 121x37; FormatPattern 999999
      ProcessValue <- "Data_AI.Hi_limit"
   IOField "I/O field_4" at 189,211 size 121x37; FormatPattern 999999
      ProcessValue <- "Data_AI.Lo_limit"
   IOField "I/O field_5" at 189,275 size 121x37; FormatPattern 999999
      ProcessValue <- "Data_AI.Lolo_limit"
   IOField "I/O field_6" at 187,336 size 121x37; FormatPattern 999999
      ProcessValue <- "Data_AI.Value_hi_scale"
   IOField "I/O field_7" at 188,389 size 121x37; FormatPattern 999999
      ProcessValue <- "Data_AI.Value_lo_scale"
   TextField "Text field_2" at 32,339 size 138x29; Text 'Шкала верх'
   TextField "Text field_3" at 32,389 size 126x29; Text 'Шкала низ'
   TextField "OBR" at 5,12 size 80x49; Text 'ОБР'
      Visibility <- "Data_AI.Lo_raw"
   TextField "KZ" at 5,12 size 80x49; Text 'КЗ'
      Visibility <- "Data_AI.Hi_raw"
*)

(* ===== HMI "SERVER1" =====

PopupScreen "hg1jahs3gd0jgsab97a9837-059c-40a0-b5d1-acf1acfc15230" 329x445
   ScreenModuleView "FP_AI_1" at 0,1 size 325x440; ScreenModuleType ""
      Guid_{11997190-26185} <- "Data_AI_Data{1}"
*)